/// GearOut parameter strucure
TYPE ST_AxisGearOutParameter :
STRUCT
	/// Halt axis after gear out
	bHaltAxis: BOOL := TRUE;
	/// Gear out (not implemented)
	stOptions: ST_GearOutOptions;
END_STRUCT
END_TYPE

(* stored: Version 1.1.0.1, ProductVersion 3.1.4022.9
   DUT ST_AxisGearOutParameter: Id {10b0e8f0-5740-413a-80ea-e58b175a566c} *)
